(* PLC project Unnamed, Unknown Unnamed 1 *)
(* stored: creationDateTime 2024-11-06T16:10:19, modificationDateTime 2024-11-07T17:48:03 *)

TYPE atatype0 : BOOL;
END_TYPE

PROGRAM Start_Stop_Control_System
  VAR
    Up_Start AT %IX0.0 : BOOL;
    Down_Stop AT %IX0.1 : BOOL;
  END_VAR
  VAR
    Latch : BOOL;
  END_VAR
  VAR
    LED AT %QX0.0 : BOOL;
  END_VAR

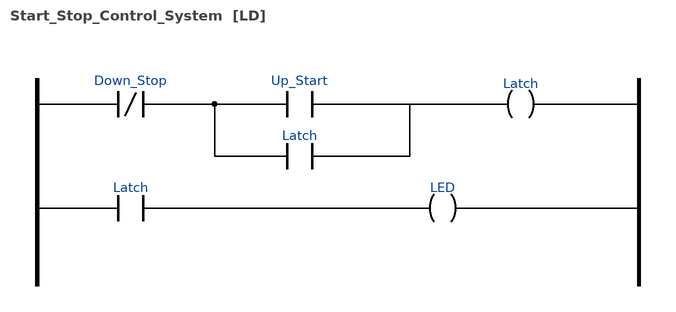
(* LD diagram, written out as Structured Text *)
LED := Latch;
Latch := NOT Down_Stop AND (Up_Start OR Latch);
END_PROGRAM

CONFIGURATION Config0
  RESOURCE Res0 ON PLC
    TASK task0(INTERVAL := T#20ms, PRIORITY := 0);
    PROGRAM instance0 WITH task0 : Start_Stop_Control_System;
  END_RESOURCE
END_CONFIGURATION
